INTERFACE I_CommandInvoker

METHOD PUBLIC CyclicLogic
END_METHOD

METHOD PUBLIC Initialise : BOOL
VAR_INPUT
  commandQueue : I_CommandQueue;
END_VAR
END_METHOD

METHOD PUBLIC Reset
END_METHOD

END_INTERFACE

(* stored: Version 1.1.0.1
   Itf I_CommandInvoker: Id {d898da51-0896-4fe7-b22b-9ec23a208296}
   Folder Methods: Id {f5b3d1ee-cb70-46f7-a281-f5c6b2c0d17f}
   Method CyclicLogic: Id {f5888847-01b4-4574-9959-4ad590fda087}
   Method Initialise: Id {9956610d-7ffe-4290-a760-4ad3c5ec748e}
   Method Reset: Id {bb1bd401-9d8f-4092-a274-b5503152378b} *)
